// TIA Portal project "自动立体仓库" (V16)

(* hardware
DEVICE "S7-1200 station_1"  S7-1200 Station
   slot 0: "Rack_0"  S7-1200 Rack  Rack  V1.0
   slot 1: "PLC_1"  CPU 1212C DC/DC/DC  6ES7 212-1AE40-0XB0  V4.2
   slot 2: "DI 16/DQ 16x24VDC_1"  6ES7 223-1BL32-0XB0  V2.0
DEVICE "GSD device_1"  GSD.Device.PN
   slot 0: "机架"  Rack  V1.0
   slot 0: "IRC5-PNIO-Device"  IRC5 PNIO-Device  0  1
      slot 0: "IRC5 PNIO-Device"  IRC5 PNIO-Device  0  1
      slot 1: "Interface1"  Interface1
         slot 1: "Port1"  Port1
   slot 1: "DI 8 bytes_1"  DI 8 bytes
      slot 0: "DI 8 bytes"  DI 8 bytes
   slot 2: "DO 8 bytes_1"  DO 8 bytes
      slot 0: "DO 8 bytes"  DO 8 bytes
*)

// ===== PLC "PLC_1"  CPU 1212C DC/DC/DC =====

VAR_GLOBAL   // PLC tag table "默认变量表"
   "System_Byte" AT %MB1 : Byte;
   "FirstScan" AT %M1.0 : Bool;
   "DiagStatusUpdate" AT %M1.1 : Bool;
   "AlwaysTRUE" AT %M1.2 : Bool;
   "AlwaysFALSE" AT %M1.3 : Bool;
   "Tag_1" AT %M8.1 : Bool;
   "Tag_3" AT %MD90 : Real;
   "Tag_4" AT %MD80 : Real;
END_VAR

VAR_GLOBAL   // PLC tag table "io表"
   "x轴脉冲" AT %Q0.0 : Bool;
   "x轴方向" AT %Q0.1 : Bool;
   "z轴脉冲" AT %Q0.2 : Bool;
   "z轴方向" AT %Q0.3 : Bool;
   "x轴前限位" AT %I0.0 : Bool;
   "x轴原点" AT %I0.1 : Bool;
   "x轴后限位" AT %I0.2 : Bool;
   "z轴上限位" AT %I0.3 : Bool;
   "z轴原点" AT %I0.4 : Bool;
   "z轴下限位" AT %I0.5 : Bool;
   "输送线A右传感器" AT %I1.0 : Bool;
   "输送线A左传感器" AT %I1.1 : Bool;
   "启动" AT %I1.4 : Bool;
   "复位" AT %I1.5 : Bool;
   "急停" AT %I1.6 : Bool;
   "单机/联动" AT %I1.7 : Bool;
   "旋转气缸左转" AT %I2.0 : Bool;
   "旋转气缸右转" AT %I2.1 : Bool;
   "伸出前限位" AT %I2.2 : Bool;
   "伸出后限位" AT %I2.3 : Bool;
   "黄灯" AT %Q1.0 : Bool;
   "红灯" AT %Q1.2 : Bool;
   "气缸左旋" AT %Q1.4 : Bool;
   "气缸右旋" AT %Q1.5 : Bool;
   "气缸伸缩" AT %Q1.6 : Bool;
   "气缸夹紧" AT %Q1.7 : Bool;
   "输送带A正转" AT %Q2.0 : Bool;
   "输送带A反转" AT %Q2.1 : Bool;
   "手自动切换" AT %M2.6 : Bool;
   "自动启动按钮" AT %M2.7 : Bool;
   "x轴前进-触点" AT %M6.0 : Bool;
   "x轴后退-触点" AT %M6.1 : Bool;
   "z轴下移-触点" AT %M6.2 : Bool;
   "z轴上移-触点" AT %M6.3 : Bool;
   "x轴前进" AT %M7.0 : Bool;
   "x轴后退" AT %M7.1 : Bool;
   "x轴回原点" AT %M7.2 : Bool;
   "z轴下移" AT %M7.3 : Bool;
   "z轴上移" AT %M7.4 : Bool;
   "z轴回原点" AT %M7.5 : Bool;
   "x轴启动标志位" AT %M2.0 : Bool;
   "x轴完成标志位" AT %M2.1 : Bool;
   "z轴启动标志位" AT %M2.2 : Bool;
   "z轴完成标志位" AT %M2.3 : Bool;
   "x轴回原点(1)" AT %M2.4 : Bool;
   "z轴回原点(1)" AT %M2.5 : Bool;
   "启动整个程序" AT %M5.0 : Bool;
   "tag_2" AT %M5.2 : Bool;
   "自动模式" AT %M5.3 : Bool;
   "x轴取料移动标志" AT %M3.0 : Bool;
   "tag_5" AT %M20.0 : Bool;
   "z轴取料移动标志位" AT %M3.1 : Bool;
   "tag_7" AT %M20.1 : Bool;
   "x轴定位数据" AT %MD30 : Real;
   "z轴定位数据" AT %MD40 : Real;
   "启动气缸左旋标志位" AT %M3.2 : Bool;
   "启动气缸伸缩标志位" AT %M3.3 : Bool;
   "启动气缸夹取标志位" AT %M3.4 : Bool;
   "z轴上升标志位" AT %M3.5 : Bool;
   "tag_12" AT %M20.2 : Bool;
   "气缸回缩标志位" AT %M3.6 : Bool;
   "气缸右旋标志位" AT %M3.7 : Bool;
   "x轴启动放料位" AT %M4.0 : Bool;
   "tag_16" AT %M20.3 : Bool;
   "z轴上升到放料位" AT %M4.1 : Bool;
   "tag_18" AT %M20.4 : Bool;
   "气缸伸出放料标志位" AT %M4.2 : Bool;
   "气缸放松放料标志位" AT %M4.3 : Bool;
   "tag_21" AT %M4.4 : Bool;
   "X轴报错复位" AT %M7.6 : Bool;
   "z轴报错复位" AT %M7.7 : Bool;
   "tag_22" AT %MD50 : Real;
   "tag_23" AT %MD60 : Real;
   "tag_24" AT %MD70 : Real;
   "绿灯" AT %Q1.1 : Bool;
END_VAR

DATA_BLOCK "公共数据"   // DB3
{ S7_Optimized_Access := 'TRUE' }
VERSION : 0.1
   VAR
      定时器 : Struct
         T1 : Array[0..20] of IEC_TIMER;
      END_STRUCT;
      自动模式 : Struct
         计数 : Array[0..6] of DInt;
         计数器 : DInt;
         自动入库的当前数据 : DInt;
         自动入库当前库有料 : Bool;
         自动入库当前库无料 : Bool;
         自动入库x距离 : Real;
         自动入库x行 : DInt;
         自动入库y列 : DInt;
         x变量 : Real;
         y变量 : Real;
      END_STRUCT;
      手动模式 : Struct
         手动入库x行 : DInt;
         手动入库y列 : DInt;
         x变量 : Real;
         y变量 : Real;
      END_STRUCT;
   END_VAR
BEGIN
END_DATA_BLOCK

DATA_BLOCK "轴_1"   // DB1, Motion_DB
{ S7_Optimized_Access := 'TRUE' }
AUTHOR : SIMATIC
FAMILY : BasicMC
NAME : TO_PosAx
VERSION : 6.0
// stored: InstanceOfName TO_PositioningAxis
"TO_PositioningAxis"
BEGIN
   // Axis.DirectionOutputEnabledCU = TRUE
   // Axis.HomingReferencePointSwitch_AddressCU = %I0.1
   // Axis.LengthUnitNormalized.Distance = 1013
   // Axis.PositionLimitsMax_AddressCU = %I0.2
   // Axis.PositionLimitsMin_AddressCU = %I0.0
   // Axis.OnlinePtoModeCU = 16#0000_0002
   // Axis.SelectedChannel2EnumCU = %Q0.1
   // Axis.SelectedChannel1EnumCU = %Q0.0
   // Pulse.MinDeltaDeltaFrequencyCU = 0.004
   // Pulse.MaxDeltaDeltaFrequencyCU = 1.0E+10
   // Pulse.MinDeltaFrequencyCU = 0.005
   // Pulse.MaxDeltaFrequencyCU = 9.5E+9
   // Pulse.MinFrequencyCU = 1.0
   // Pulse.MaxFrequencyCU = 100000.0
   // Pulse.OutputSourceCU = 16#0000_0000
   // Axis.SelectPTO = 0
END_DATA_BLOCK

DATA_BLOCK "轴_2"   // DB2, Motion_DB
{ S7_Optimized_Access := 'TRUE' }
AUTHOR : SIMATIC
FAMILY : BasicMC
NAME : TO_PosAx
VERSION : 6.0
// stored: InstanceOfName TO_PositioningAxis
"TO_PositioningAxis"
BEGIN
   // Axis.DirectionOutputEnabledCU = TRUE
   // Axis.HomingReferencePointSwitch_AddressCU = %I0.4
   // Axis.LengthUnitNormalized.Distance = 1013
   // Axis.PositionLimitsMax_AddressCU = %I0.5
   // Axis.PositionLimitsMin_AddressCU = %I0.3
   // Axis.OnlinePtoModeCU = 16#0000_0002
   // Axis.SelectedChannel2EnumCU = %Q0.3
   // Axis.SelectedChannel1EnumCU = %Q0.2
   // Pulse.MinDeltaDeltaFrequencyCU = 0.004
   // Pulse.MaxDeltaDeltaFrequencyCU = 1.0E+10
   // Pulse.MinDeltaFrequencyCU = 0.005
   // Pulse.MaxDeltaFrequencyCU = 9.5E+9
   // Pulse.MinFrequencyCU = 1.0
   // Pulse.MaxFrequencyCU = 100000.0
   // Pulse.OutputSourceCU = 16#0000_0000
   // Axis.SelectPTO = 1
   // Axis.OnlinePtoIndexCU = 1
END_DATA_BLOCK

FUNCTION "电机运转" : Void   // FC1, LAD
{ S7_Optimized_Access := 'TRUE' }
VERSION : 0.1
BEGIN

REGION Network 1: 启动两个电机轴
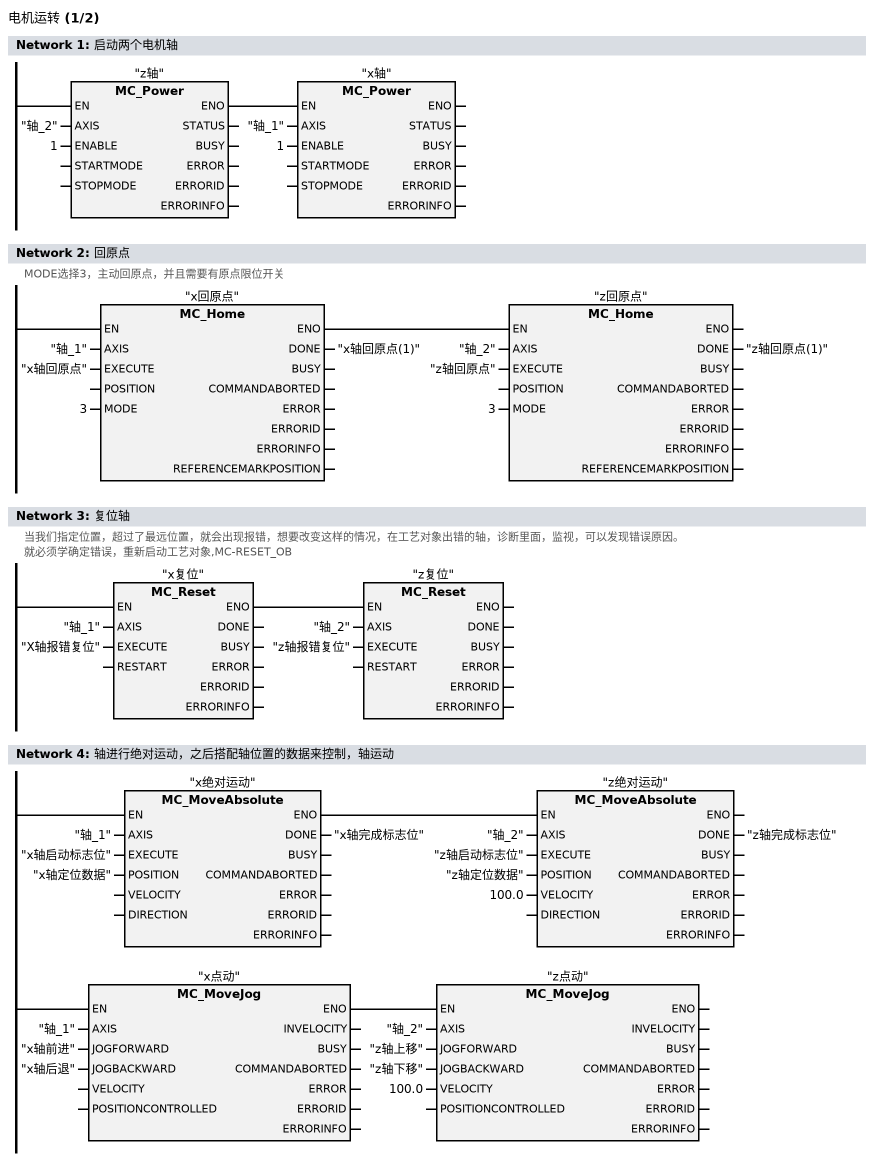
   // ENO of a box is taken as its EN; it also drops when the box reports an error
   "z轴"(Axis := "轴_2", Enable := 1);   // MC_Power
   "x轴"(Axis := "轴_1", Enable := 1);   // MC_Power
END_REGION

REGION Network 2: 回原点
   // MODE选择3，主动回原点，并且需要有原点限位开关
   // ENO of a box is taken as its EN; it also drops when the box reports an error
   "x回原点"(Axis := "轴_1", Execute := "x轴回原点", Mode := 3, Done => "x轴回原点(1)");   // MC_Home
   "z回原点"(Axis := "轴_2", Execute := "z轴回原点", Mode := 3, Done => "z轴回原点(1)");   // MC_Home
END_REGION

REGION Network 3: 复位轴
   // 当我们指定位置，超过了最远位置，就会出现报错，想要改变这样的情况，在工艺对象出错的轴，诊断里面，监视，可以发现错误原因。
   // 就必须学确定错误，重新启动工艺对象,MC-RESET_OB
   // ENO of a box is taken as its EN; it also drops when the box reports an error
   "x复位"(Axis := "轴_1", Execute := "X轴报错复位");   // MC_Reset
   "z复位"(Axis := "轴_2", Execute := "z轴报错复位");   // MC_Reset
END_REGION

REGION Network 4: 轴进行绝对运动，之后搭配轴位置的数据来控制，轴运动
   // ENO of a box is taken as its EN; it also drops when the box reports an error
   "x绝对运动"(Axis := "轴_1", Execute := "x轴启动标志位", Position := "x轴定位数据", Done => "x轴完成标志位");   // MC_MoveAbsolute
   "z绝对运动"(Axis := "轴_2", Execute := "z轴启动标志位", Position := "z轴定位数据", Velocity := 100.0, Done => "z轴完成标志位");   // MC_MoveAbsolute
   "x点动"(Axis := "轴_1", JogForward := "x轴前进", JogBackward := "x轴后退");   // MC_MoveJog
   "z点动"(Axis := "轴_2", JogForward := "z轴上移", JogBackward := "z轴下移", Velocity := 100.0);   // MC_MoveJog
END_REGION

REGION Network 5
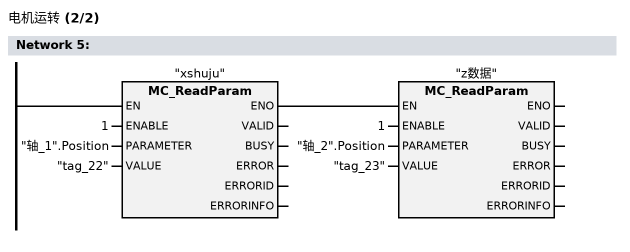
   // ENO of a box is taken as its EN; it also drops when the box reports an error
   "xshuju"(Enable := 1, Parameter := "轴_1".Position, Value := "tag_22");   // MC_ReadParam
   "z数据"(Enable := 1, Parameter := "轴_2".Position, Value := "tag_23");   // MC_ReadParam
END_REGION
END_FUNCTION

FUNCTION "自动模式运行" : Void   // FC2, LAD
{ S7_Optimized_Access := 'TRUE' }
VERSION : 0.1
   VAR_TEMP   // added for the SCL form of the ladder/FBD networks
      _w1 : Bool;
      _w2 : Bool;
      _w3 : Bool;
      _w4 : Bool;
      _w5 : Bool;
      _w6 : Bool;
   END_VAR
BEGIN

REGION Network 1: 启动，电机回原点
   // 这里是先开启回原点，之后用x，z轴的数值来判断是否达到原点，然后再复位回原点的程序，之后启动运输物料，在这之前应该写一个，abb程序用来将物料运输到传送带上
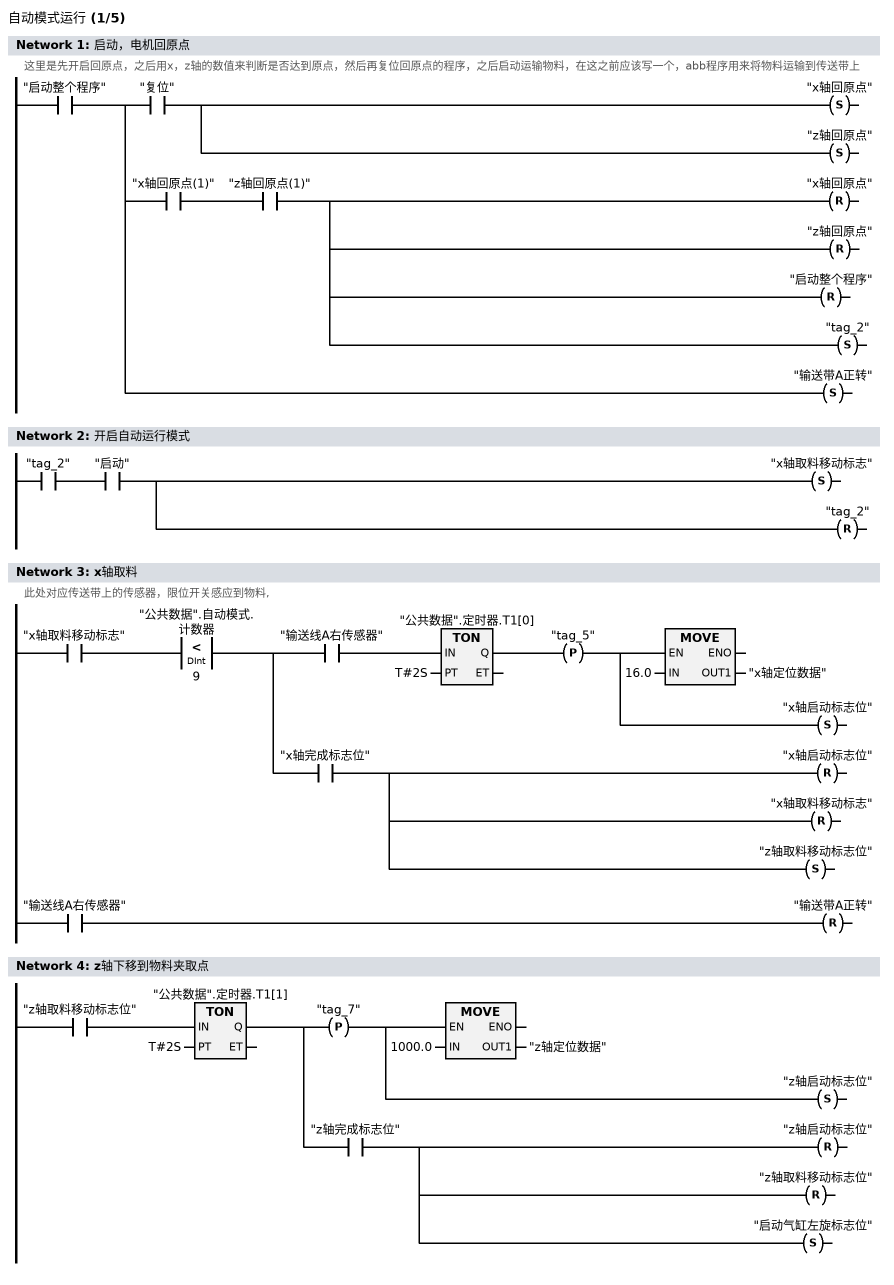
   RUNG wire#powerrail
      Contact( "启动整个程序" )
      wire#w1
      Contact( "复位" )
      wire#w2
      S_Coil( "x轴回原点" )
   END_RUNG
   RUNG wire#w2
      S_Coil( "z轴回原点" )
   END_RUNG
   RUNG wire#w1
      Contact( "x轴回原点(1)" )
      Contact( "z轴回原点(1)" )
      wire#w3
      R_Coil( "x轴回原点" )
   END_RUNG
   RUNG wire#w3
      R_Coil( "z轴回原点" )
   END_RUNG
   RUNG wire#w3
      R_Coil( "启动整个程序" )
   END_RUNG
   RUNG wire#w3
      S_Coil( "tag_2" )
   END_RUNG
   RUNG wire#w1
      S_Coil( "输送带A正转" )
   END_RUNG
   // the same network as SCL:
   IF "启动整个程序" AND "复位" THEN
       "x轴回原点" := TRUE;
       "z轴回原点" := TRUE;
   END_IF;
   IF "启动整个程序" AND "x轴回原点(1)" AND "z轴回原点(1)" THEN
       "x轴回原点" := FALSE;
       "z轴回原点" := FALSE;
   END_IF;
   #_w1 := "启动整个程序";
   #_w2 := "启动整个程序" AND "x轴回原点(1)" AND "z轴回原点(1)";
   IF #_w2 THEN
       "启动整个程序" := FALSE;
       "tag_2" := TRUE;
   END_IF;
   IF #_w1 THEN "输送带A正转" := TRUE; END_IF;
END_REGION

REGION Network 2: 开启自动运行模式
   RUNG wire#powerrail
      Contact( "tag_2" )
      Contact( "启动" )
      wire#w1
      S_Coil( "x轴取料移动标志" )
   END_RUNG
   RUNG wire#w1
      R_Coil( "tag_2" )
   END_RUNG
   // the same network as SCL:
   IF "tag_2" AND "启动" THEN
       "x轴取料移动标志" := TRUE;
       "tag_2" := FALSE;
   END_IF;
END_REGION

REGION Network 3: x轴取料
   // 此处对应传送带上的传感器，限位开关感应到物料,
   #_w1 := "x轴取料移动标志" AND ("公共数据".自动模式.计数器 < 9);
   "公共数据".定时器.T1[0].TON(IN := #_w1 AND "输送线A右传感器", PT := T#2S);
   #_w2 := "公共数据".定时器.T1[0].Q AND NOT "tag_5";   // rising edge
   "tag_5" := "公共数据".定时器.T1[0].Q;
   IF #_w2 THEN
       "x轴定位数据" := 16.0;
       "x轴启动标志位" := TRUE;
   END_IF;
   IF #_w1 AND "x轴完成标志位" THEN
       "x轴启动标志位" := FALSE;
       "x轴取料移动标志" := FALSE;
       "z轴取料移动标志位" := TRUE;
   END_IF;
   IF "输送线A右传感器" THEN "输送带A正转" := FALSE; END_IF;
END_REGION

REGION Network 4: z轴下移到物料夹取点
   "公共数据".定时器.T1[1].TON(IN := "z轴取料移动标志位", PT := T#2S);
   #_w1 := "公共数据".定时器.T1[1].Q AND NOT "tag_7";   // rising edge
   "tag_7" := "公共数据".定时器.T1[1].Q;
   IF #_w1 THEN
       "z轴定位数据" := 1000.0;
       "z轴启动标志位" := TRUE;
   END_IF;
   IF "公共数据".定时器.T1[1].Q AND "z轴完成标志位" THEN
       "z轴启动标志位" := FALSE;
       "z轴取料移动标志位" := FALSE;
       "启动气缸左旋标志位" := TRUE;
   END_IF;
END_REGION

REGION Network 5: 启动气缸左旋回来物料
   // 因为气缸，可能上次完成之后，气缸没有旋转回来
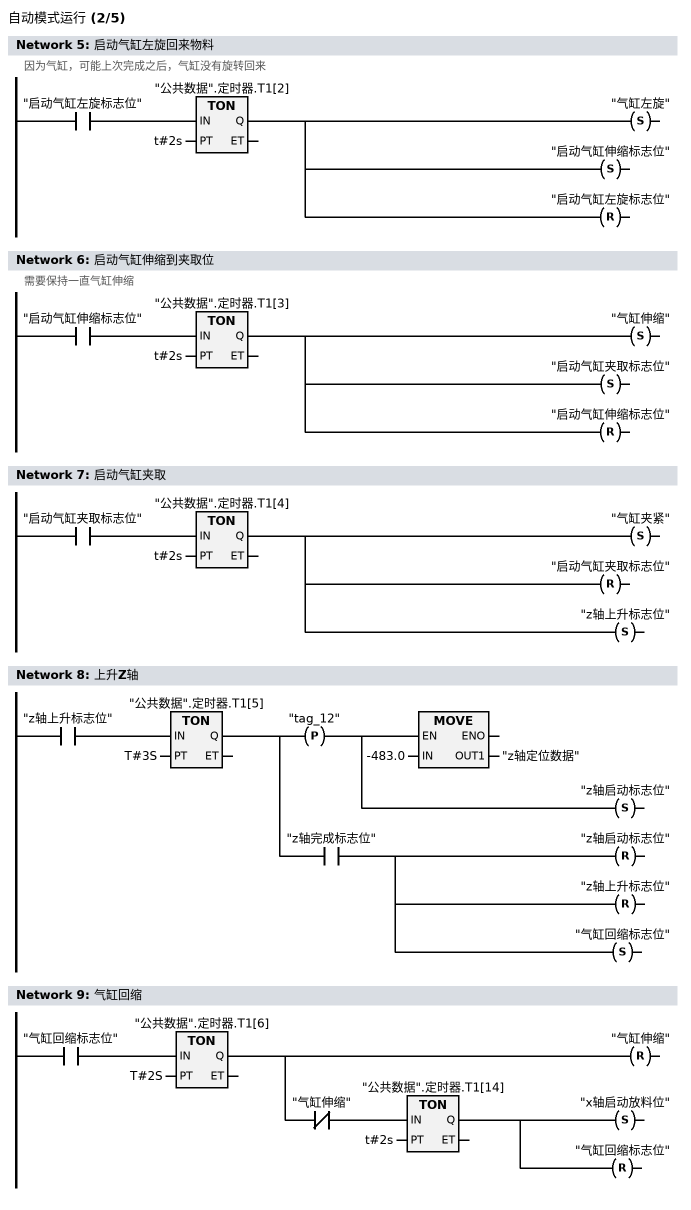
   "公共数据".定时器.T1[2].TON(IN := "启动气缸左旋标志位", PT := t#2s);
   IF "公共数据".定时器.T1[2].Q THEN
       "气缸左旋" := TRUE;
       "启动气缸伸缩标志位" := TRUE;
       "启动气缸左旋标志位" := FALSE;
   END_IF;
END_REGION

REGION Network 6: 启动气缸伸缩到夹取位
   // 需要保持一直气缸伸缩
   "公共数据".定时器.T1[3].TON(IN := "启动气缸伸缩标志位", PT := t#2s);
   IF "公共数据".定时器.T1[3].Q THEN
       "气缸伸缩" := TRUE;
       "启动气缸夹取标志位" := TRUE;
       "启动气缸伸缩标志位" := FALSE;
   END_IF;
END_REGION

REGION Network 7: 启动气缸夹取
   "公共数据".定时器.T1[4].TON(IN := "启动气缸夹取标志位", PT := t#2s);
   IF "公共数据".定时器.T1[4].Q THEN
       "气缸夹紧" := TRUE;
       "启动气缸夹取标志位" := FALSE;
       "z轴上升标志位" := TRUE;
   END_IF;
END_REGION

REGION Network 8: 上升Z轴
   "公共数据".定时器.T1[5].TON(IN := "z轴上升标志位", PT := T#3S);
   #_w1 := "公共数据".定时器.T1[5].Q AND NOT "tag_12";   // rising edge
   "tag_12" := "公共数据".定时器.T1[5].Q;
   IF #_w1 THEN
       "z轴定位数据" := -483.0;
       "z轴启动标志位" := TRUE;
   END_IF;
   IF "公共数据".定时器.T1[5].Q AND "z轴完成标志位" THEN
       "z轴启动标志位" := FALSE;
       "z轴上升标志位" := FALSE;
       "气缸回缩标志位" := TRUE;
   END_IF;
END_REGION

REGION Network 9: 气缸回缩
   "公共数据".定时器.T1[6].TON(IN := "气缸回缩标志位", PT := T#2S);
   IF "公共数据".定时器.T1[6].Q THEN "气缸伸缩" := FALSE; END_IF;
   "公共数据".定时器.T1[14].TON(IN := "公共数据".定时器.T1[6].Q AND NOT "气缸伸缩", PT := t#2s);
   IF "公共数据".定时器.T1[14].Q THEN
       "x轴启动放料位" := TRUE;
       "气缸回缩标志位" := FALSE;
   END_IF;
END_REGION

REGION Network 10: x轴移动到放料位，每排放三个，之后开始循环，之后有对y开始运动
   // 我对于x轴来说，每排放3个，
   // 所以当我想要进行循环的时候，我可以写一个递增的数据，每当x移动3次之后
   // 就在z轴上升的程序里面，进行一次加法/减法计算
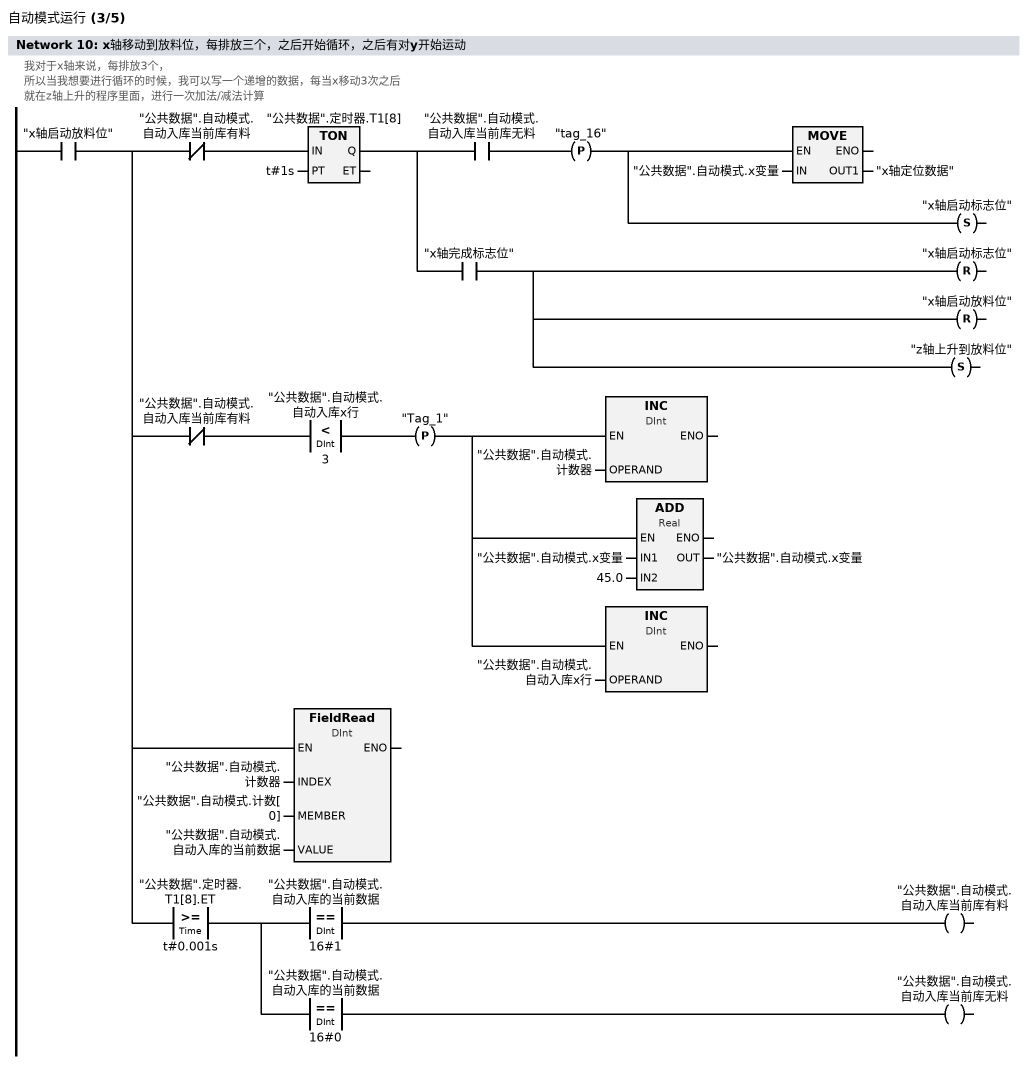
   // no SCL statement known for FieldRead: written as a call
   "公共数据".定时器.T1[8].TON(IN := "x轴启动放料位" AND NOT "公共数据".自动模式.自动入库当前库有料, PT := t#1s);
   #_w1 := "公共数据".定时器.T1[8].Q AND "公共数据".自动模式.自动入库当前库无料;
   #_w2 := #_w1 AND NOT "tag_16";   // rising edge
   "tag_16" := #_w1;
   IF #_w2 THEN
       "x轴定位数据" := "公共数据".自动模式.x变量;
       "x轴启动标志位" := TRUE;
   END_IF;
   IF "公共数据".定时器.T1[8].Q AND "x轴完成标志位" THEN "x轴启动标志位" := FALSE; END_IF;
   #_w3 := "x轴启动放料位";
   IF "公共数据".定时器.T1[8].Q AND "x轴完成标志位" THEN
       "x轴启动放料位" := FALSE;
       "z轴上升到放料位" := TRUE;
   END_IF;
   #_w4 := #_w3 AND NOT "公共数据".自动模式.自动入库当前库有料 AND ("公共数据".自动模式.自动入库x行 < 3);
   #_w5 := #_w4 AND NOT "Tag_1";   // rising edge
   "Tag_1" := #_w4;
   IF #_w5 THEN
       "公共数据".自动模式.计数器 := "公共数据".自动模式.计数器 + 1;
       "公共数据".自动模式.x变量 := "公共数据".自动模式.x变量 + 45.0;
       "公共数据".自动模式.自动入库x行 := "公共数据".自动模式.自动入库x行 + 1;
   END_IF;
   IF #_w3 THEN
       FieldRead(index := "公共数据".自动模式.计数器, member := "公共数据".自动模式.计数[0], value := "公共数据".自动模式.自动入库的当前数据);
   END_IF;
   #_w6 := #_w3 AND ("公共数据".定时器.T1[8].ET >= t#0.001s);
   "公共数据".自动模式.自动入库当前库有料 := #_w6 AND ("公共数据".自动模式.自动入库的当前数据 = 16#1);
   "公共数据".自动模式.自动入库当前库无料 := #_w6 AND ("公共数据".自动模式.自动入库的当前数据 = 16#0);
END_REGION

REGION Network 11: Z轴放置到放料位上方
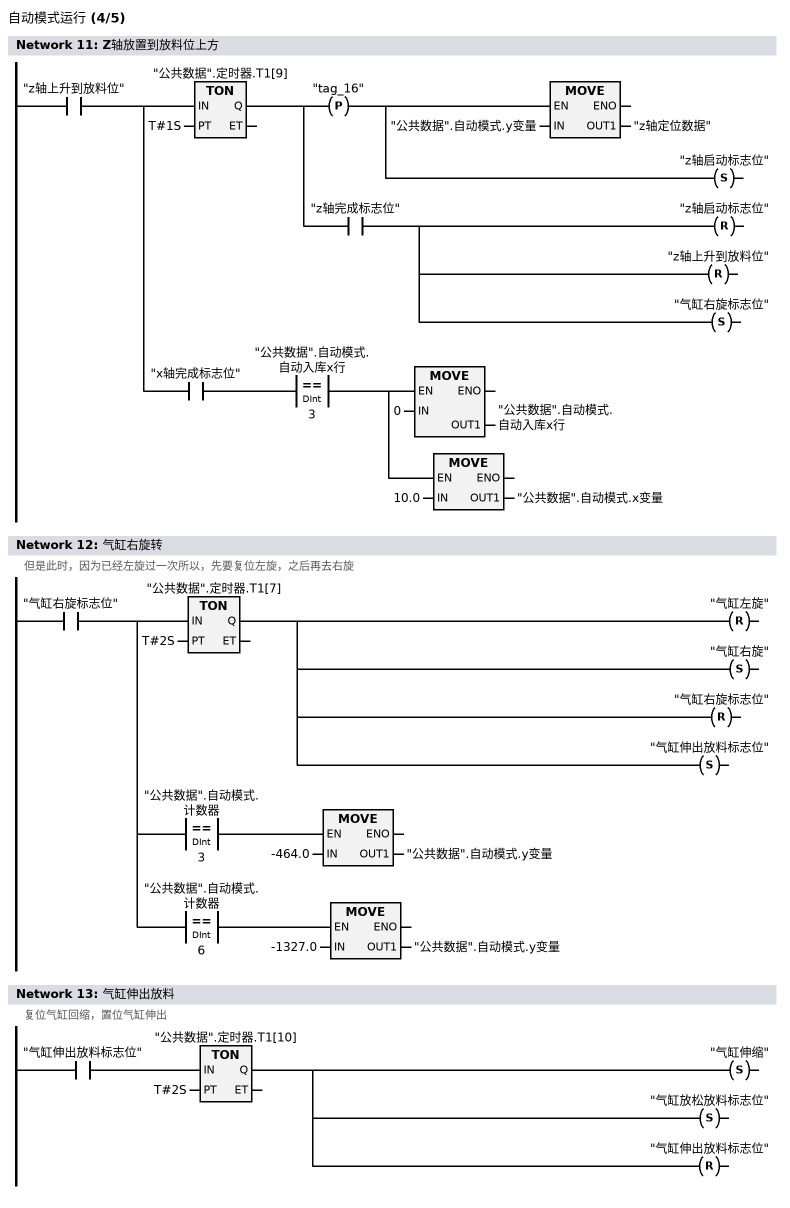
   "公共数据".定时器.T1[9].TON(IN := "z轴上升到放料位", PT := T#1S);
   #_w1 := "公共数据".定时器.T1[9].Q AND NOT "tag_16";   // rising edge
   "tag_16" := "公共数据".定时器.T1[9].Q;
   IF #_w1 THEN
       "z轴定位数据" := "公共数据".自动模式.y变量;
       "z轴启动标志位" := TRUE;
   END_IF;
   IF "公共数据".定时器.T1[9].Q AND "z轴完成标志位" THEN "z轴启动标志位" := FALSE; END_IF;
   #_w2 := "z轴上升到放料位";
   IF "公共数据".定时器.T1[9].Q AND "z轴完成标志位" THEN
       "z轴上升到放料位" := FALSE;
       "气缸右旋标志位" := TRUE;
   END_IF;
   #_w3 := #_w2 AND "x轴完成标志位" AND ("公共数据".自动模式.自动入库x行 = 3);
   IF #_w3 THEN
       "公共数据".自动模式.自动入库x行 := 0;
       "公共数据".自动模式.x变量 := 10.0;
   END_IF;
END_REGION

REGION Network 12: 气缸右旋转
   // 但是此时，因为已经左旋过一次所以，先要复位左旋，之后再去右旋
   "公共数据".定时器.T1[7].TON(IN := "气缸右旋标志位", PT := T#2S);
   IF "公共数据".定时器.T1[7].Q THEN
       "气缸左旋" := FALSE;
       "气缸右旋" := TRUE;
   END_IF;
   #_w1 := "气缸右旋标志位";
   IF "公共数据".定时器.T1[7].Q THEN
       "气缸右旋标志位" := FALSE;
       "气缸伸出放料标志位" := TRUE;
   END_IF;
   IF #_w1 AND ("公共数据".自动模式.计数器 = 3) THEN "公共数据".自动模式.y变量 := -464.0; END_IF;
   IF #_w1 AND ("公共数据".自动模式.计数器 = 6) THEN "公共数据".自动模式.y变量 := -1327.0; END_IF;
END_REGION

REGION Network 13: 气缸伸出放料
   // 复位气缸回缩，置位气缸伸出
   "公共数据".定时器.T1[10].TON(IN := "气缸伸出放料标志位", PT := T#2S);
   IF "公共数据".定时器.T1[10].Q THEN
       "气缸伸缩" := TRUE;
       "气缸放松放料标志位" := TRUE;
       "气缸伸出放料标志位" := FALSE;
   END_IF;
END_REGION

REGION Network 14: 夹爪松开
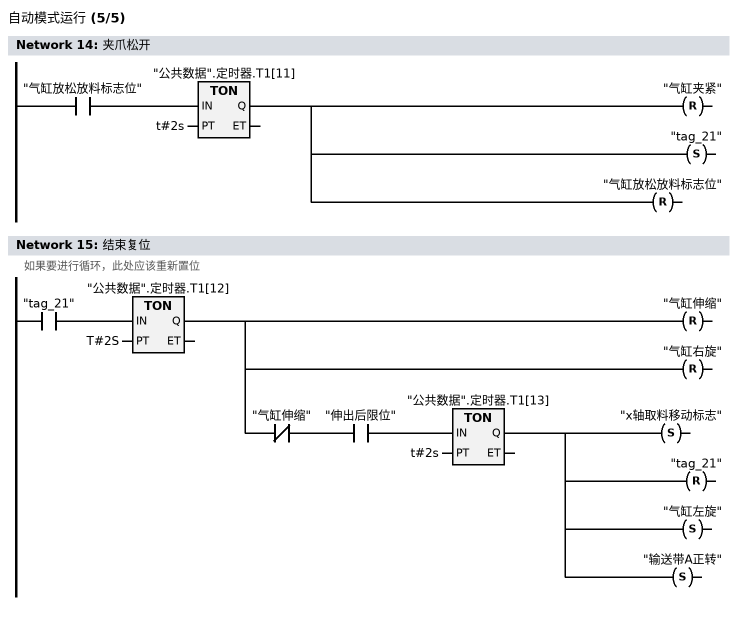
   "公共数据".定时器.T1[11].TON(IN := "气缸放松放料标志位", PT := t#2s);
   IF "公共数据".定时器.T1[11].Q THEN
       "气缸夹紧" := FALSE;
       "tag_21" := TRUE;
       "气缸放松放料标志位" := FALSE;
   END_IF;
END_REGION

REGION Network 15: 结束复位
   // 如果要进行循环，此处应该重新置位
   "公共数据".定时器.T1[12].TON(IN := "tag_21", PT := T#2S);
   IF "公共数据".定时器.T1[12].Q THEN
       "气缸伸缩" := FALSE;
       "气缸右旋" := FALSE;
   END_IF;
   "公共数据".定时器.T1[13].TON(IN := "公共数据".定时器.T1[12].Q AND NOT "气缸伸缩" AND "伸出后限位", PT := t#2s);
   IF "公共数据".定时器.T1[13].Q THEN
       "x轴取料移动标志" := TRUE;
       "tag_21" := FALSE;
       "气缸左旋" := TRUE;
       "输送带A正转" := TRUE;
   END_IF;
END_REGION
END_FUNCTION

FUNCTION "手动运行模式" : Void   // FC3, LAD
{ S7_Optimized_Access := 'TRUE' }
VERSION : 0.1
   VAR_TEMP   // added for the SCL form of the ladder/FBD networks
      _w1 : Bool;
   END_VAR
BEGIN

REGION Network 1: 初始化程序，并且启动程序
   // 利用M1.0达到首次循环，启动复位
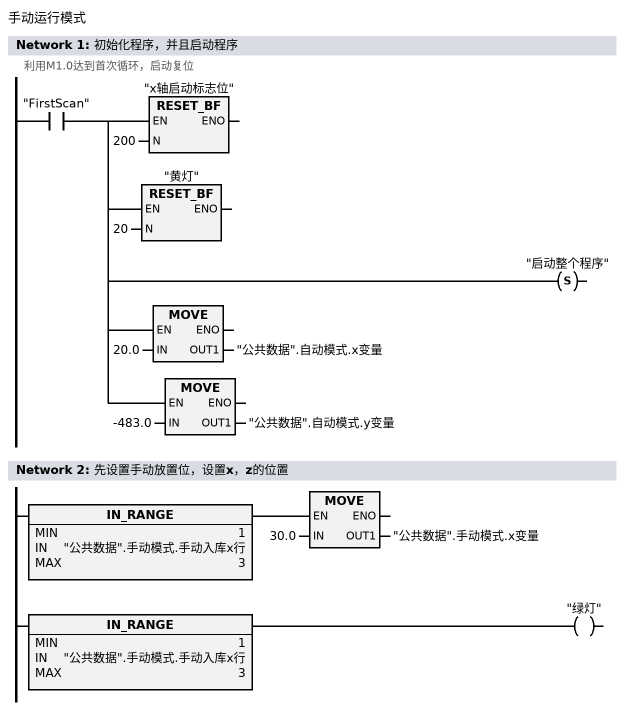
   // no SCL statement known for RBitfield: written as a call
   #_w1 := "FirstScan";
   IF #_w1 THEN
       RESET_BF(operand := "x轴启动标志位", n := 200);
       RESET_BF(operand := "黄灯", n := 20);
       "启动整个程序" := TRUE;
       "公共数据".自动模式.x变量 := 20.0;
       "公共数据".自动模式.y变量 := -483.0;
   END_IF;
END_REGION

REGION Network 2: 先设置手动放置位，设置x，z的位置
   RUNG wire#powerrail
      { S7_Templates := "SrcType := DInt" } InRange(min := 1, in := "公共数据".手动模式.手动入库x行, max := 3)
      Move(in := 30.0, out1 => "公共数据".手动模式.x变量)
   END_RUNG
   RUNG wire#powerrail
      { S7_Templates := "SrcType := DInt" } InRange(min := 1, in := "公共数据".手动模式.手动入库x行, max := 3)
      Coil( "绿灯" )
   END_RUNG
   // the same network as SCL:
   IF (1 <= "公共数据".手动模式.手动入库x行) AND ("公共数据".手动模式.手动入库x行 <= 3) THEN "公共数据".手动模式.x变量 := 30.0; END_IF;
   "绿灯" := (1 <= "公共数据".手动模式.手动入库x行) AND ("公共数据".手动模式.手动入库x行 <= 3);
END_REGION
END_FUNCTION

ORGANIZATION_BLOCK "Main"   // OB1, LAD, ProgramCycle
TITLE = "Main Program Sweep (Cycle)"
{ S7_Optimized_Access := 'TRUE' }
VERSION : 0.1
   VAR_INPUT
      Initial_Call : Bool;   // Initial call of this OB
      Remanence : Bool;   // =True, if remanent data are available
   END_VAR
   VAR_TEMP   // added for the SCL form of the ladder/FBD networks
      _w1 : Bool;
   END_VAR
BEGIN

REGION Network 1: 初始化程序，并且启动程序
   // 利用M1.0达到首次循环，启动复位
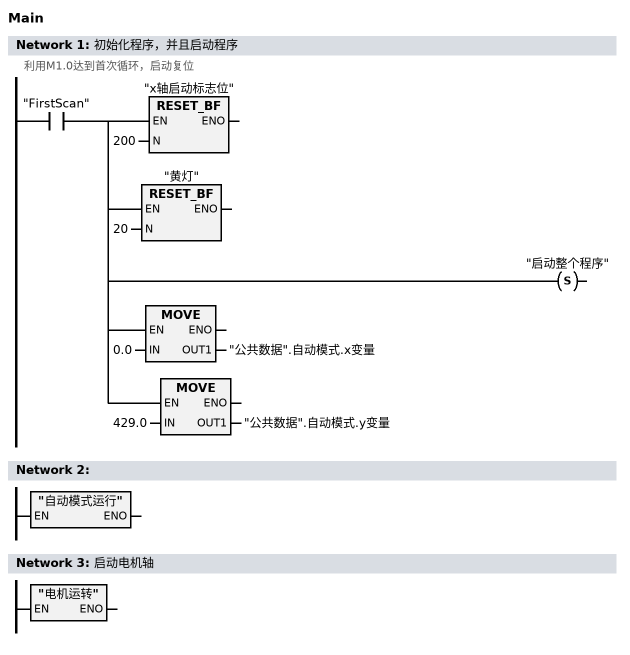
   // no SCL statement known for RBitfield: written as a call
   #_w1 := "FirstScan";
   IF #_w1 THEN
       RESET_BF(operand := "x轴启动标志位", n := 200);
       RESET_BF(operand := "黄灯", n := 20);
       "启动整个程序" := TRUE;
       "公共数据".自动模式.x变量 := 0.0;
       "公共数据".自动模式.y变量 := 429.0;
   END_IF;
END_REGION

REGION Network 2
   RUNG wire#powerrail
      "自动模式运行"()
   END_RUNG
   // the same network as SCL:
   "自动模式运行"();
END_REGION

REGION Network 3: 启动电机轴
   RUNG wire#powerrail
      "电机运转"()
   END_RUNG
   // the same network as SCL:
   "电机运转"();
END_REGION
END_ORGANIZATION_BLOCK